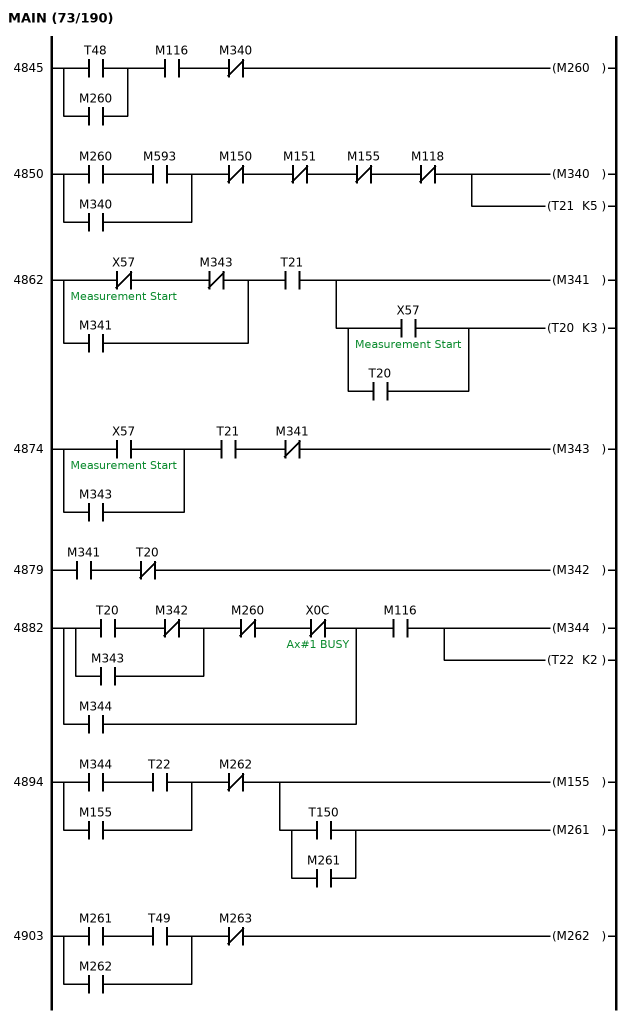
[picture p72: ladder of MAIN, rungs at steps 4845 to 4903]
4845  LD      T48
      OR      M260
      AND     M116
      ANI     M340
      OUT     M260
4850  LD      M260
      AND     M593
      OR      M340
      ANI     M150
      ANI     M151
      ANI     M155
      ANI     M118
      OUT     M340
      OUT     T21 K5
4862  LDI     X57  ; Measurement Start
      ANI     M343
      OR      M341
      AND     T21
      OUT     M341
      LD      X57  ; Measurement Start
      OR      T20
      ANB
      OUT     T20 K3
4874  LD      X57  ; Measurement Start
      OR      M343
      AND     T21
      ANI     M341
      OUT     M343
4879  LD      M341
      ANI     T20
      OUT     M342
4882  LD      T20
      ANI     M342
      OR      M343
      ANI     M260
      ANI     X0C  ; Ax#1 BUSY
      OR      M344
      AND     M116
      OUT     M344
      OUT     T22 K2
4894  LD      M344
      AND     T22
      OR      M155
      ANI     M262
      OUT     M155
      LD      T150
      OR      M261
      ANB
      OUT     M261
4903  LD      M261
      AND     T49
      OR      M262
      ANI     M263
      OUT     M262
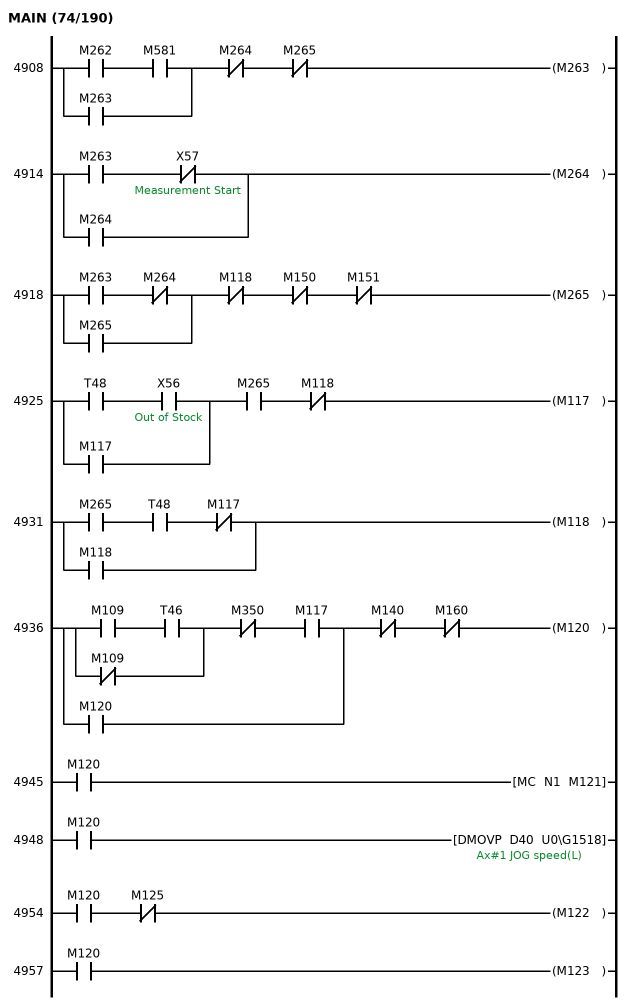
4908  LD      M262
      AND     M581
      OR      M263
      ANI     M264
      ANI     M265
      OUT     M263
4914  LD      M263
      ANI     X57  ; Measurement Start
      OR      M264
      OUT     M264
4918  LD      M263
      ANI     M264
      OR      M265
      ANI     M118
      ANI     M150
      ANI     M151
      OUT     M265
4925  LD      T48
      AND     X56  ; Out of Stock
      OR      M117
      AND     M265
      ANI     M118
      OUT     M117
4931  LD      M265
      AND     T48
      ANI     M117
      OR      M118
      OUT     M118
4936  LD      M109
      AND     T46
      ORI     M109
      ANI     M350
      AND     M117
      OR      M120
      ANI     M140
      ANI     M160
      OUT     M120
4945  LD      M120
      MC      N1 M121
4948  LD      M120
      DMOVP   D40 U0\G1518
4954  LD      M120
      ANI     M125
      OUT     M122
4957  LD      M120
      OUT     M123
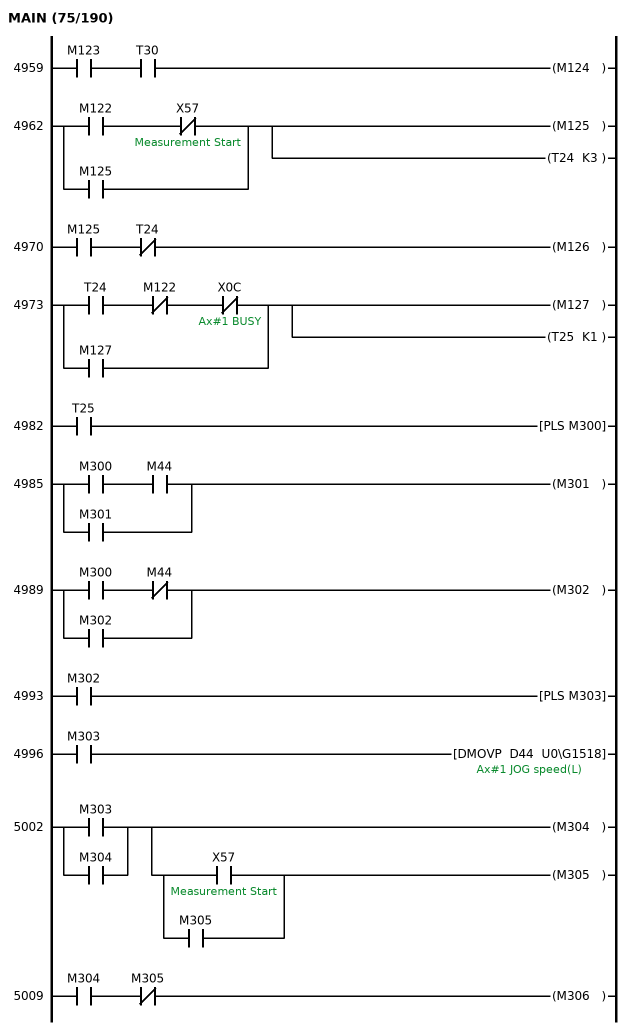
4959  LD      M123
      AND     T30
      OUT     M124
4962  LD      M122
      ANI     X57  ; Measurement Start
      OR      M125
      OUT     M125
      OUT     T24 K3
4970  LD      M125
      ANI     T24
      OUT     M126
4973  LD      T24
      ANI     M122
      ANI     X0C  ; Ax#1 BUSY
      OR      M127
      OUT     M127
      OUT     T25 K1
4982  LD      T25
      PLS     M300
4985  LD      M300
      AND     M44
      OR      M301
      OUT     M301
4989  LD      M300
      ANI     M44
      OR      M302
      OUT     M302
4993  LD      M302
      PLS     M303
4996  LD      M303
      DMOVP   D44 U0\G1518
5002  LD      M303
      OR      M304
      OUT     M304
      LD      X57  ; Measurement Start
      OR      M305
      ANB
      OUT     M305
5009  LD      M304
      ANI     M305
      OUT     M306
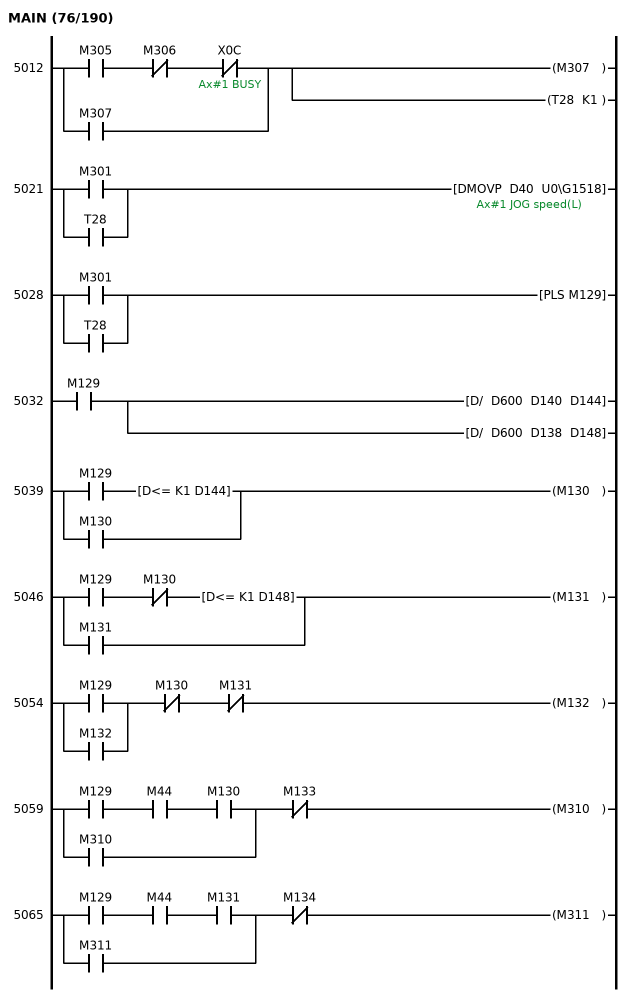
5012  LD      M305
      ANI     M306
      ANI     X0C  ; Ax#1 BUSY
      OR      M307
      OUT     M307
      OUT     T28 K1
5021  LD      M301
      OR      T28
      DMOVP   D40 U0\G1518
5028  LD      M301
      OR      T28
      PLS     M129
5032  LD      M129
      D/      D600 D140 D144
      D/      D600 D138 D148
5039  LD      M129
      ANDD<=  K1 D144
      OR      M130
      OUT     M130
5046  LD      M129
      ANI     M130
      ANDD<=  K1 D148
      OR      M131
      OUT     M131
5054  LD      M129
      OR      M132
      ANI     M130
      ANI     M131
      OUT     M132
5059  LD      M129
      AND     M44
      AND     M130
      OR      M310
      ANI     M133
      OUT     M310
5065  LD      M129
      AND     M44
      AND     M131
      OR      M311
      ANI     M134
      OUT     M311
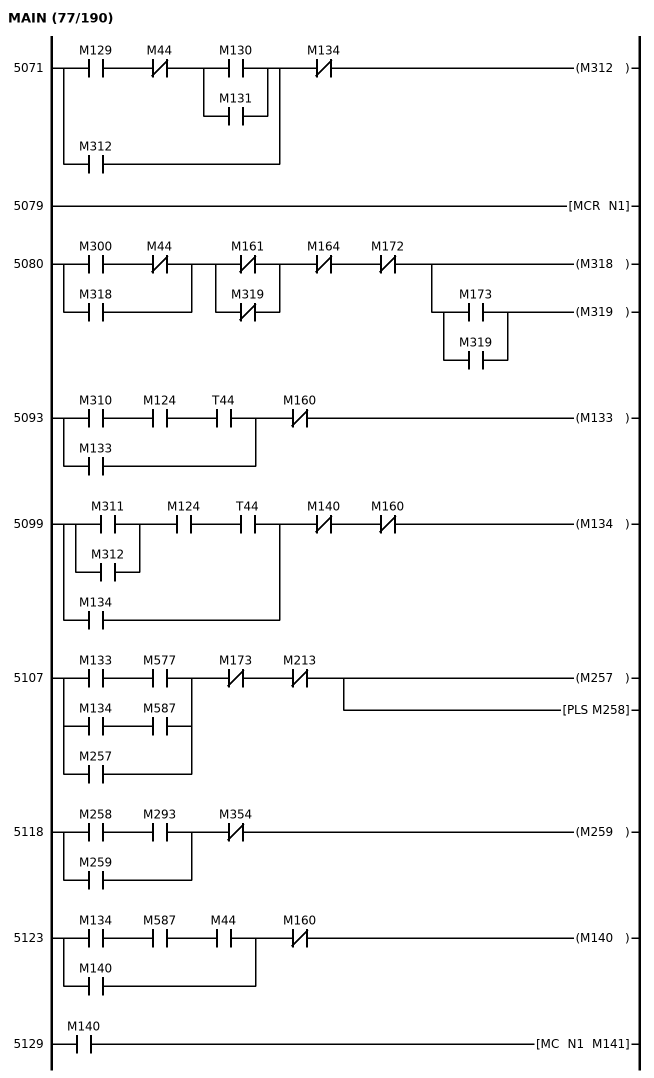
5071  LD      M129
      ANI     M44
      LD      M130
      OR      M131
      ANB
      OR      M312
      ANI     M134
      OUT     M312
5079  MCR     N1
5080  LD      M300
      ANI     M44
      OR      M318
      LDI     M161
      ORI     M319
      ANB
      ANI     M164
      ANI     M172
      OUT     M318
      LD      M173
      OR      M319
      ANB
      OUT     M319
5093  LD      M310
      AND     M124
      AND     T44
      OR      M133
      ANI     M160
      OUT     M133
5099  LD      M311
      OR      M312
      AND     M124
      AND     T44
      OR      M134
      ANI     M140
      ANI     M160
      OUT     M134
5107  LD      M133
      AND     M577
      LD      M134
      AND     M587
      ORB
      OR      M257
      ANI     M173
      ANI     M213
      OUT     M257
      PLS     M258
5118  LD      M258
      AND     M293
      OR      M259
      ANI     M354
      OUT     M259
5123  LD      M134
      AND     M587
      AND     M44
      OR      M140
      ANI     M160
      OUT     M140
5129  LD      M140
      MC      N1 M141
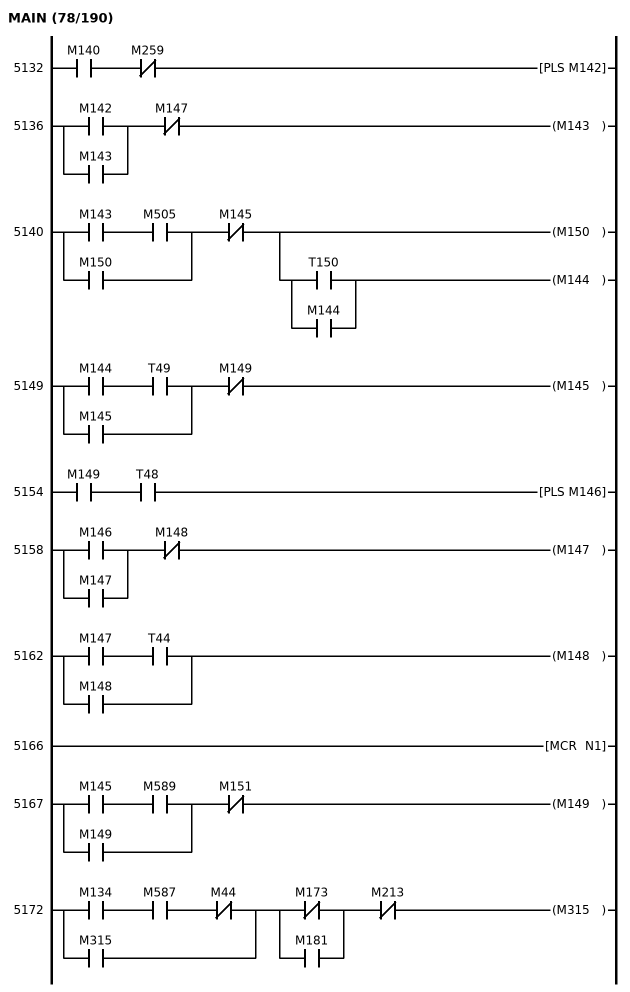
5132  LD      M140
      ANI     M259
      PLS     M142
5136  LD      M142
      OR      M143
      ANI     M147
      OUT     M143
5140  LD      M143
      AND     M505
      OR      M150
      ANI     M145
      OUT     M150
      LD      T150
      OR      M144
      ANB
      OUT     M144
5149  LD      M144
      AND     T49
      OR      M145
      ANI     M149
      OUT     M145
5154  LD      M149
      AND     T48
      PLS     M146
5158  LD      M146
      OR      M147
      ANI     M148
      OUT     M147
5162  LD      M147
      AND     T44
      OR      M148
      OUT     M148
5166  MCR     N1
5167  LD      M145
      AND     M589
      OR      M149
      ANI     M151
      OUT     M149
5172  LD      M134
      AND     M587
      ANI     M44
      OR      M315
      LDI     M173
      OR      M181
      ANB
      ANI     M213
      OUT     M315
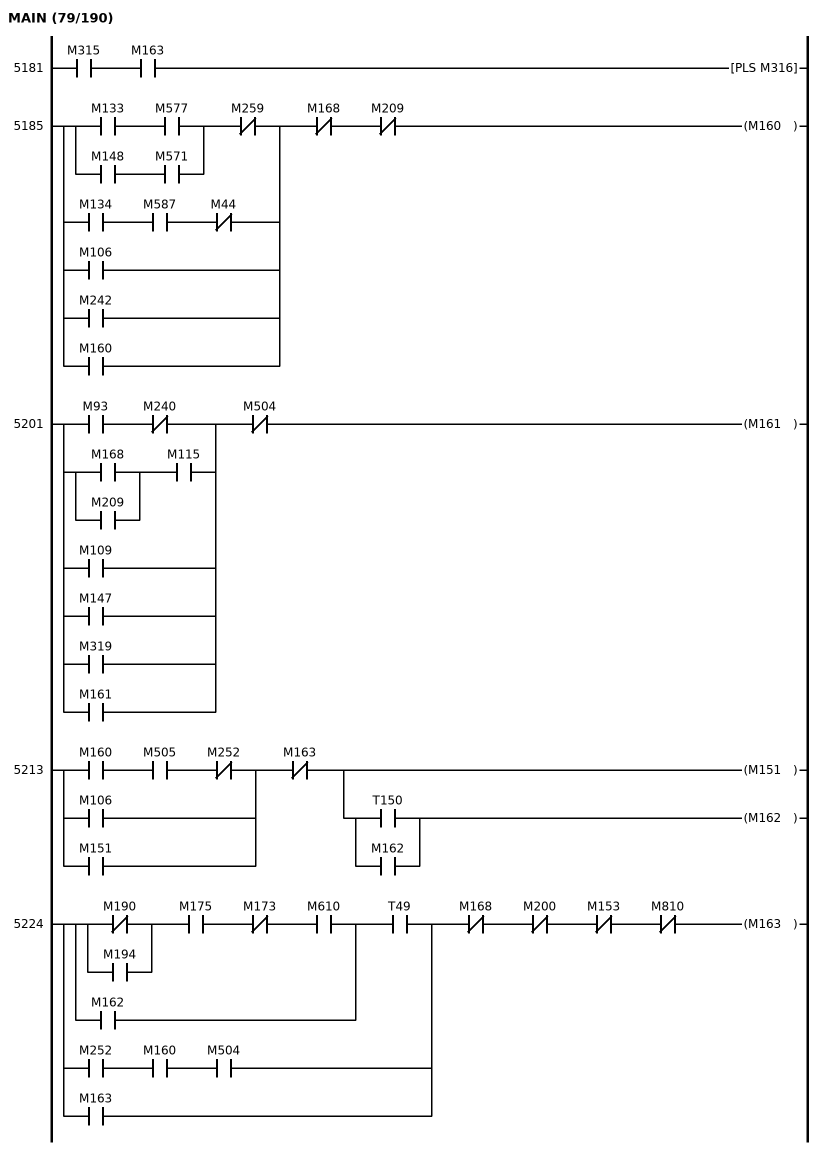
5181  LD      M315
      AND     M163
      PLS     M316
5185  LD      M133
      AND     M577
      LD      M148
      AND     M571
      ORB
      ANI     M259
      LD      M134
      AND     M587
      ANI     M44
      ORB
      OR      M106
      OR      M242
      OR      M160
      ANI     M168
      ANI     M209
      OUT     M160
5201  LD      M93
      ANI     M240
      LD      M168
      OR      M209
      AND     M115
      ORB
      OR      M109
      OR      M147
      OR      M319
      OR      M161
      ANI     M504
      OUT     M161
5213  LD      M160
      AND     M505
      ANI     M252
      OR      M106
      OR      M151
      ANI     M163
      OUT     M151
      LD      T150
      OR      M162
      ANB
      OUT     M162
5224  LDI     M190
      OR      M194
      AND     M175
      ANI     M173
      AND     M610
      OR      M162
      AND     T49
      LD      M252
      AND     M160
      AND     M504
      ORB
      OR      M163
      ANI     M168
      ANI     M200
      ANI     M153
      ANI     M810
      OUT     M163
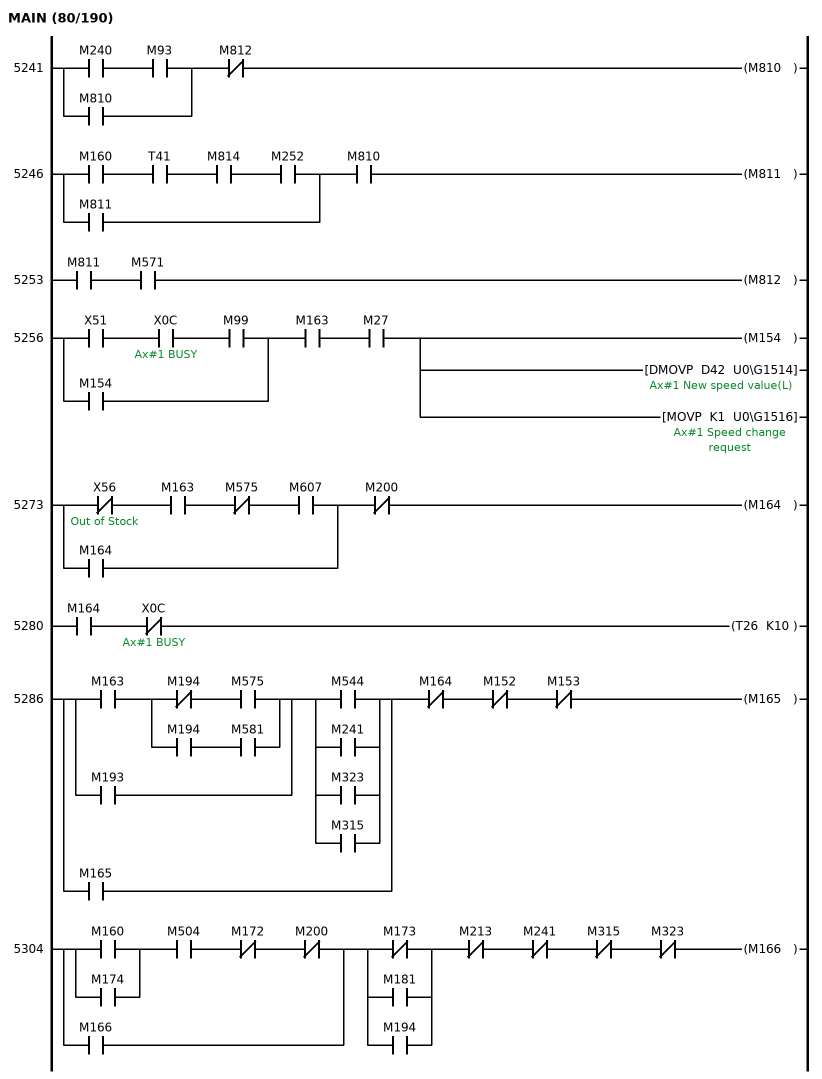
5241  LD      M240
      AND     M93
      OR      M810
      ANI     M812
      OUT     M810
5246  LD      M160
      AND     T41
      AND     M814
      AND     M252
      OR      M811
      AND     M810
      OUT     M811
5253  LD      M811
      AND     M571
      OUT     M812
5256  LD      X51
      AND     X0C  ; Ax#1 BUSY
      AND     M99
      OR      M154
      AND     M163
      AND     M27
      OUT     M154
      DMOVP   D42 U0\G1514  ; Ax#1 New speed value(L)
      MOVP    K1 U0\G1516  ; Ax#1 Speed change request
5273  LDI     X56  ; Out of Stock
      AND     M163
      ANI     M575
      AND     M607
      OR      M164
      ANI     M200
      OUT     M164
5280  LD      M164
      ANI     X0C  ; Ax#1 BUSY
      OUT     T26 K10
5286  LD      M163
      LDI     M194
      AND     M575
      LD      M194
      AND     M581
      ORB
      ANB
      OR      M193
      LD      M544
      OR      M241
      OR      M323
      OR      M315
      ANB
      OR      M165
      ANI     M164
      ANI     M152
      ANI     M153
      OUT     M165
5304  LD      M160
      OR      M174
      AND     M504
      ANI     M172
      ANI     M200
      OR      M166
      LDI     M173
      OR      M181
      OR      M194
      ANB
      ANI     M213
      ANI     M241
      ANI     M315
      ANI     M323
      OUT     M166
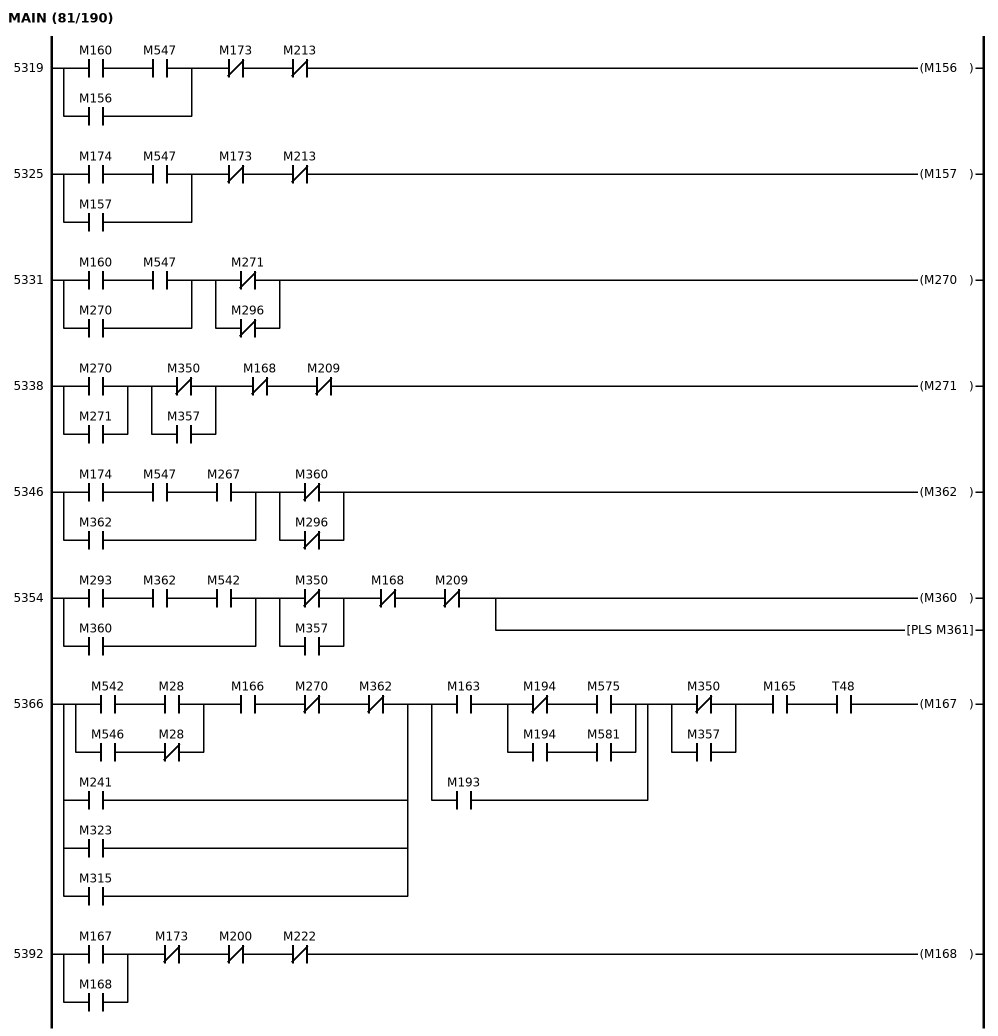
5319  LD      M160
      AND     M547
      OR      M156
      ANI     M173
      ANI     M213
      OUT     M156
5325  LD      M174
      AND     M547
      OR      M157
      ANI     M173
      ANI     M213
      OUT     M157
5331  LD      M160
      AND     M547
      OR      M270
      LDI     M271
      ORI     M296
      ANB
      OUT     M270
5338  LD      M270
      OR      M271
      LDI     M350
      OR      M357
      ANB
      ANI     M168
      ANI     M209
      OUT     M271
5346  LD      M174
      AND     M547
      AND     M267
      OR      M362
      LDI     M360
      ORI     M296
      ANB
      OUT     M362
5354  LD      M293
      AND     M362
      AND     M542
      OR      M360
      LDI     M350
      OR      M357
      ANB
      ANI     M168
      ANI     M209
      OUT     M360
      PLS     M361
5366  LD      M542
      AND     M28
      LD      M546
      ANI     M28
      ORB
      AND     M166
      ANI     M270
      ANI     M362
      OR      M241
      OR      M323
      OR      M315
      LD      M163
      LDI     M194
      AND     M575
      LD      M194
      AND     M581
      ORB
      ANB
      OR      M193
      ANB
      LDI     M350
      OR      M357
      ANB
      AND     M165
      AND     T48
      OUT     M167
5392  LD      M167
      OR      M168
      ANI     M173
      ANI     M200
      ANI     M222
      OUT     M168
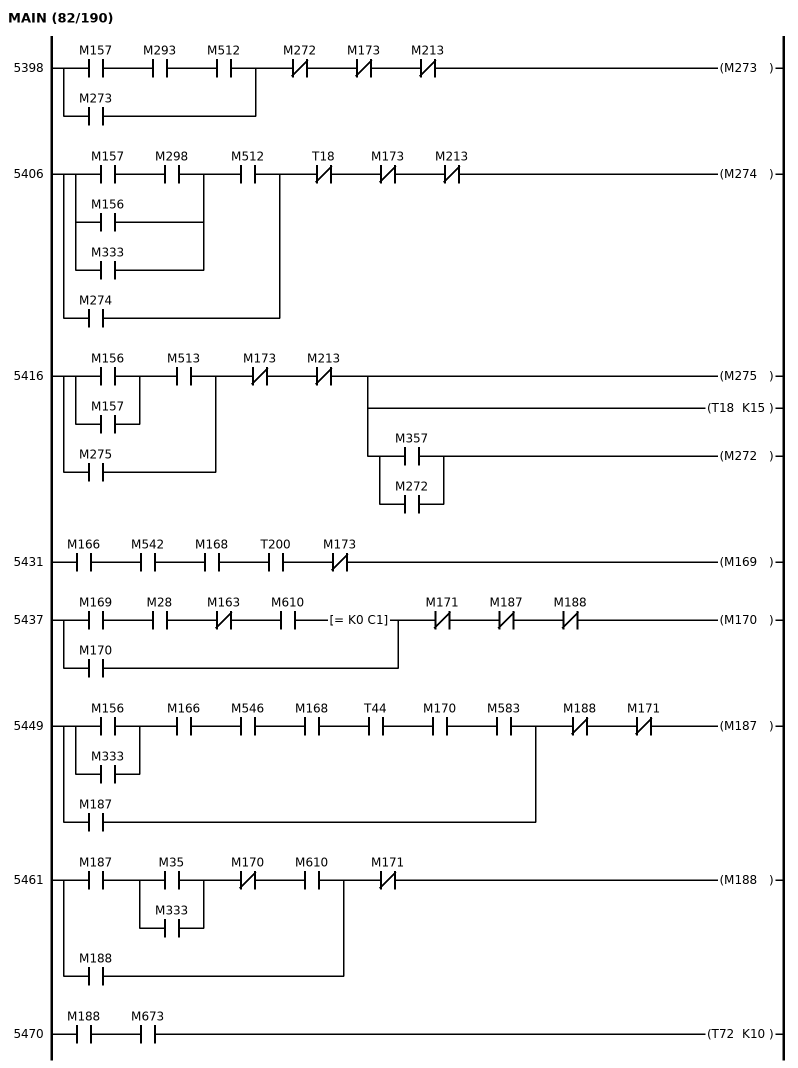
5398  LD      M157
      AND     M293
      AND     M512
      OR      M273
      ANI     M272
      ANI     M173
      ANI     M213
      OUT     M273
5406  LD      M157
      AND     M298
      OR      M156
      OR      M333
      AND     M512
      OR      M274
      ANI     T18
      ANI     M173
      ANI     M213
      OUT     M274
5416  LD      M156
      OR      M157
      AND     M513
      OR      M275
      ANI     M173
      ANI     M213
      OUT     M275
      OUT     T18 K15
      LD      M357
      OR      M272
      ANB
      OUT     M272
5431  LD      M166
      AND     M542
      AND     M168
      AND     T200
      ANI     M173
      OUT     M169
5437  LD      M169
      AND     M28
      ANI     M163
      AND     M610
      AND=    K0 C1
      OR      M170
      ANI     M171
      ANI     M187
      ANI     M188
      OUT     M170
5449  LD      M156
      OR      M333
      AND     M166
      AND     M546
      AND     M168
      AND     T44
      AND     M170
      AND     M583
      OR      M187
      ANI     M188
      ANI     M171
      OUT     M187
5461  LD      M187
      LD      M35
      OR      M333
      ANB
      ANI     M170
      AND     M610
      OR      M188
      ANI     M171
      OUT     M188
5470  LD      M188
      AND     M673
      OUT     T72 K10
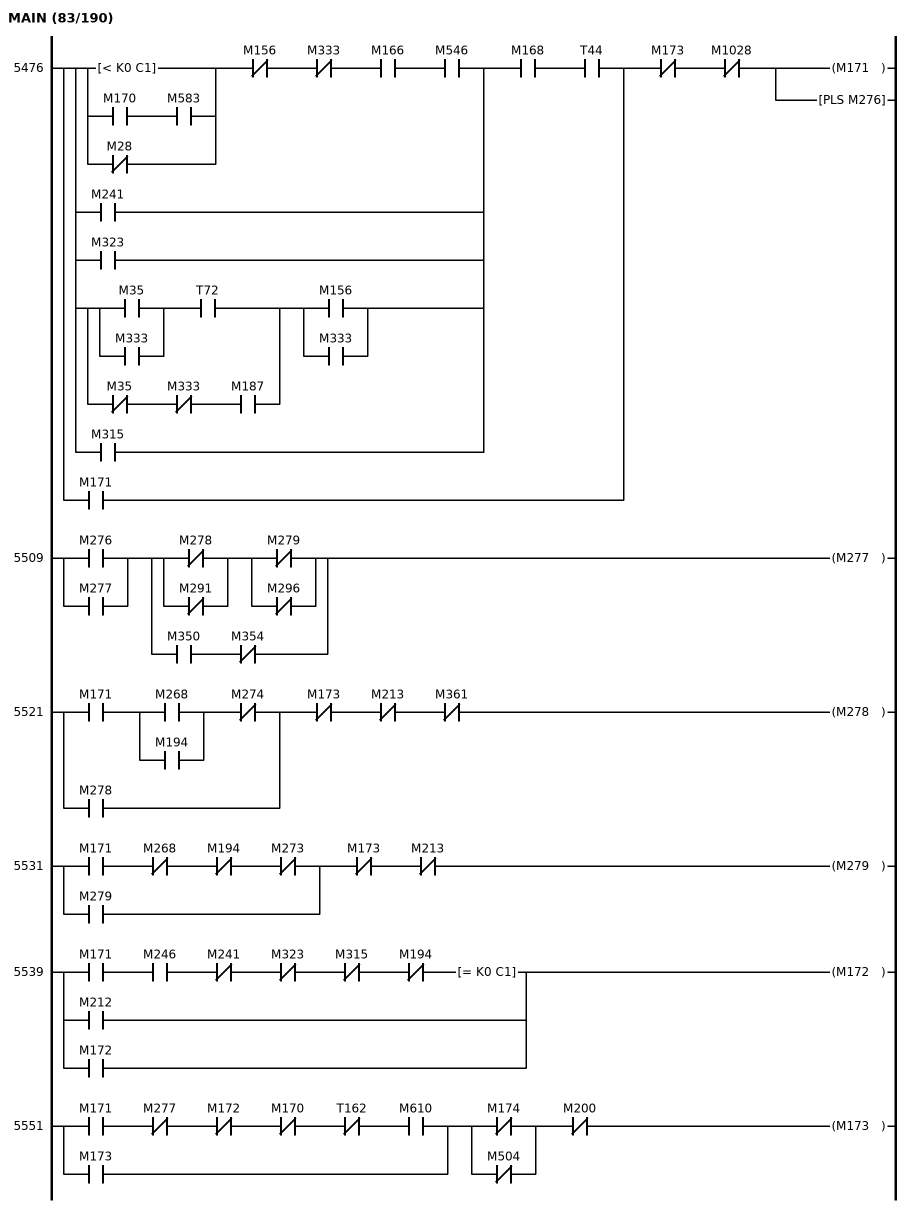
5476  LD<     K0 C1
      LD      M170
      AND     M583
      ORB
      ORI     M28
      ANI     M156
      ANI     M333
      AND     M166
      AND     M546
      OR      M241
      OR      M323
      LD      M35
      OR      M333
      AND     T72
      LDI     M35
      ANI     M333
      AND     M187
      ORB
      LD      M156
      OR      M333
      ANB
      ORB
      OR      M315
      AND     M168
      AND     T44
      OR      M171
      ANI     M173
      ANI     M1028
      OUT     M171
      PLS     M276
5509  LD      M276
      OR      M277
      LDI     M278
      ORI     M291
      LDI     M279
      ORI     M296
      ANB
      LD      M350
      ANI     M354
      ORB
      ANB
      OUT     M277
5521  LD      M171
      LD      M268
      OR      M194
      ANB
      ANI     M274
      OR      M278
      ANI     M173
      ANI     M213
      ANI     M361
      OUT     M278
5531  LD      M171
      ANI     M268
      ANI     M194
      ANI     M273
      OR      M279
      ANI     M173
      ANI     M213
      OUT     M279
5539  LD      M171
      AND     M246
      ANI     M241
      ANI     M323
      ANI     M315
      ANI     M194
      AND=    K0 C1
      OR      M212
      OR      M172
      OUT     M172
5551  LD      M171
      ANI     M277
      ANI     M172
      ANI     M170
      ANI     T162
      AND     M610
      OR      M173
      LDI     M174
      ORI     M504
      ANB
      ANI     M200
      OUT     M173
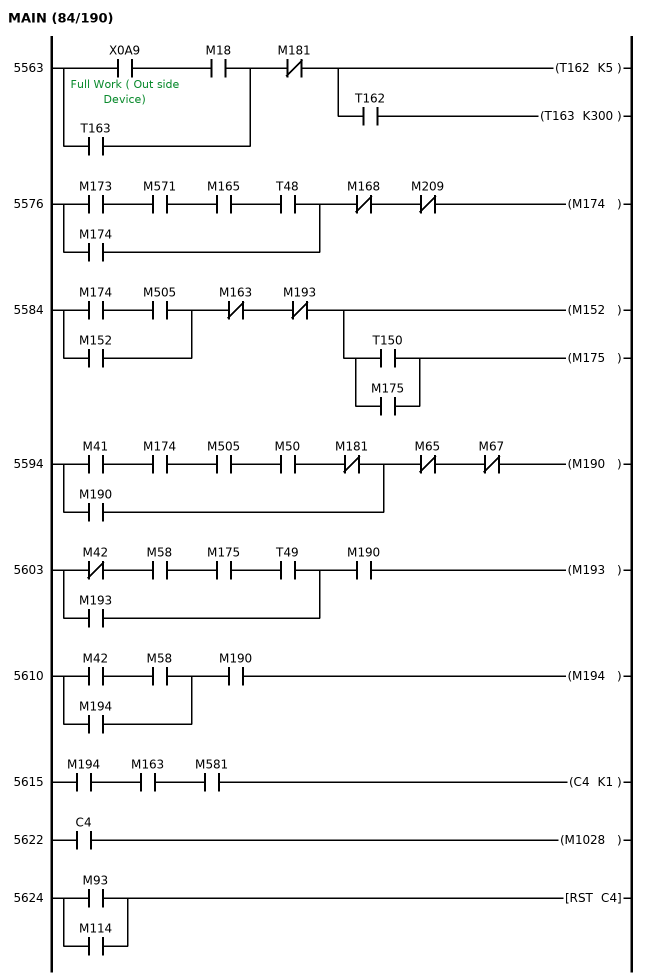
5563  LD      X0A9  ; Full Work ( Out side Device)
      AND     M18
      OR      T163
      ANI     M181
      OUT     T162 K5
      AND     T162
      OUT     T163 K300
5576  LD      M173
      AND     M571
      AND     M165
      AND     T48
      OR      M174
      ANI     M168
      ANI     M209
      OUT     M174
5584  LD      M174
      AND     M505
      OR      M152
      ANI     M163
      ANI     M193
      OUT     M152
      LD      T150
      OR      M175
      ANB
      OUT     M175
5594  LD      M41
      AND     M174
      AND     M505
      AND     M50
      ANI     M181
      OR      M190
      ANI     M65
      ANI     M67
      OUT     M190
5603  LDI     M42
      AND     M58
      AND     M175
      AND     T49
      OR      M193
      AND     M190
      OUT     M193
5610  LD      M42
      AND     M58
      OR      M194
      AND     M190
      OUT     M194
5615  LD      M194
      AND     M163
      AND     M581
      OUT     C4 K1
5622  LD      C4
      OUT     M1028
5624  LD      M93
      OR      M114
      RST     C4
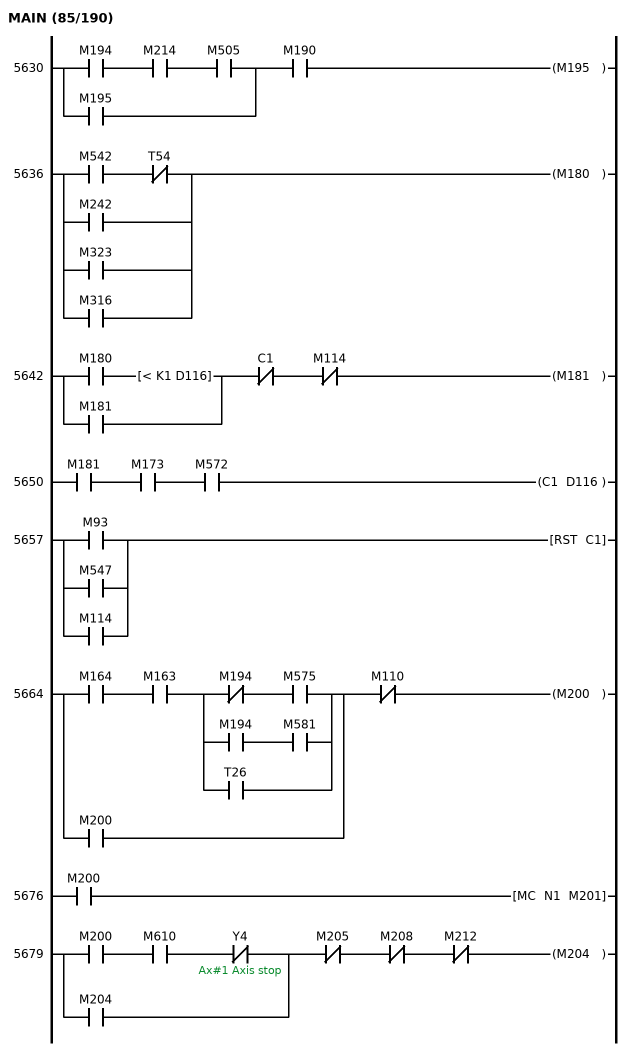
5630  LD      M194
      AND     M214
      AND     M505
      OR      M195
      AND     M190
      OUT     M195
5636  LD      M542
      ANI     T54
      OR      M242
      OR      M323
      OR      M316
      OUT     M180
5642  LD      M180
      AND<    K1 D116
      OR      M181
      ANI     C1
      ANI     M114
      OUT     M181
5650  LD      M181
      AND     M173
      AND     M572
      OUT     C1 D116
5657  LD      M93
      OR      M547
      OR      M114
      RST     C1
5664  LD      M164
      AND     M163
      LDI     M194
      AND     M575
      LD      M194
      AND     M581
      ORB
      OR      T26
      ANB
      OR      M200
      ANI     M110
      OUT     M200
5676  LD      M200
      MC      N1 M201
5679  LD      M200
      AND     M610
      ANI     Y4  ; Ax#1 Axis stop
      OR      M204
      ANI     M205
      ANI     M208
      ANI     M212
      OUT     M204
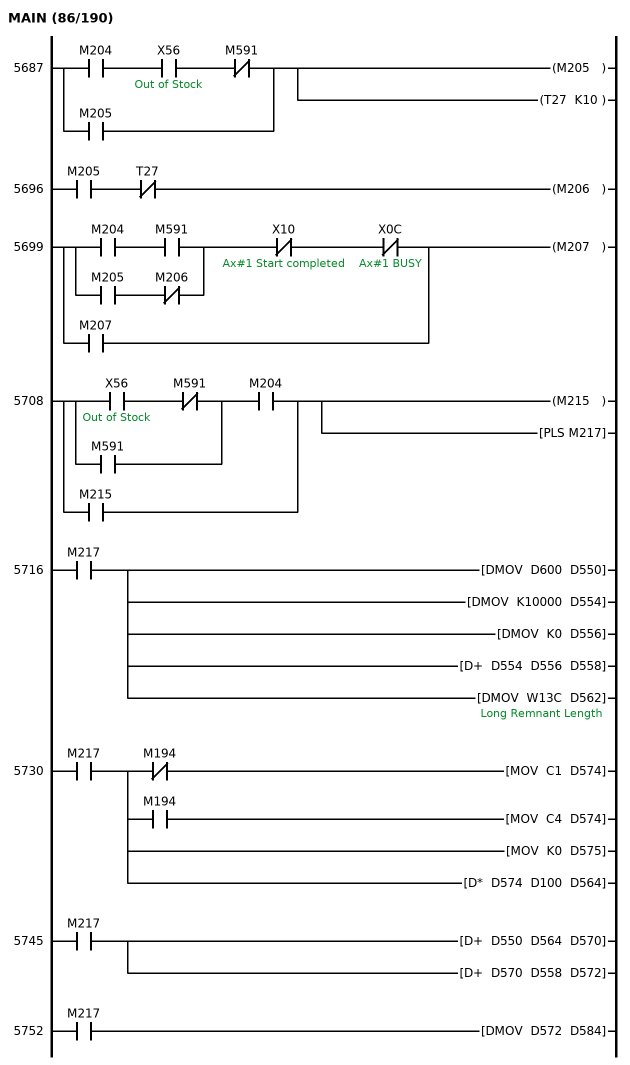
5687  LD      M204
      AND     X56  ; Out of Stock
      ANI     M591
      OR      M205
      OUT     M205
      OUT     T27 K10
5696  LD      M205
      ANI     T27
      OUT     M206
5699  LD      M204
      AND     M591
      LD      M205
      ANI     M206
      ORB
      ANI     X10  ; Ax#1 Start completed
      ANI     X0C  ; Ax#1 BUSY
      OR      M207
      OUT     M207
5708  LD      X56  ; Out of Stock
      ANI     M591
      OR      M591
      AND     M204
      OR      M215
      OUT     M215
      PLS     M217
5716  LD      M217
      DMOV    D600 D550
      DMOV    K10000 D554
      DMOV    K0 D556
      D+      D554 D556 D558
      DMOV    W13C D562  ; Long Remnant Length
5730  LD      M217
      MPS
      ANI     M194
      MOV     C1 D574
      MRD
      AND     M194
      MOV     C4 D574
      MPP
      MOV     K0 D575
      D*      D574 D100 D564
5745  LD      M217
      D+      D550 D564 D570
      D+      D570 D558 D572
5752  LD      M217
      DMOV    D572 D584
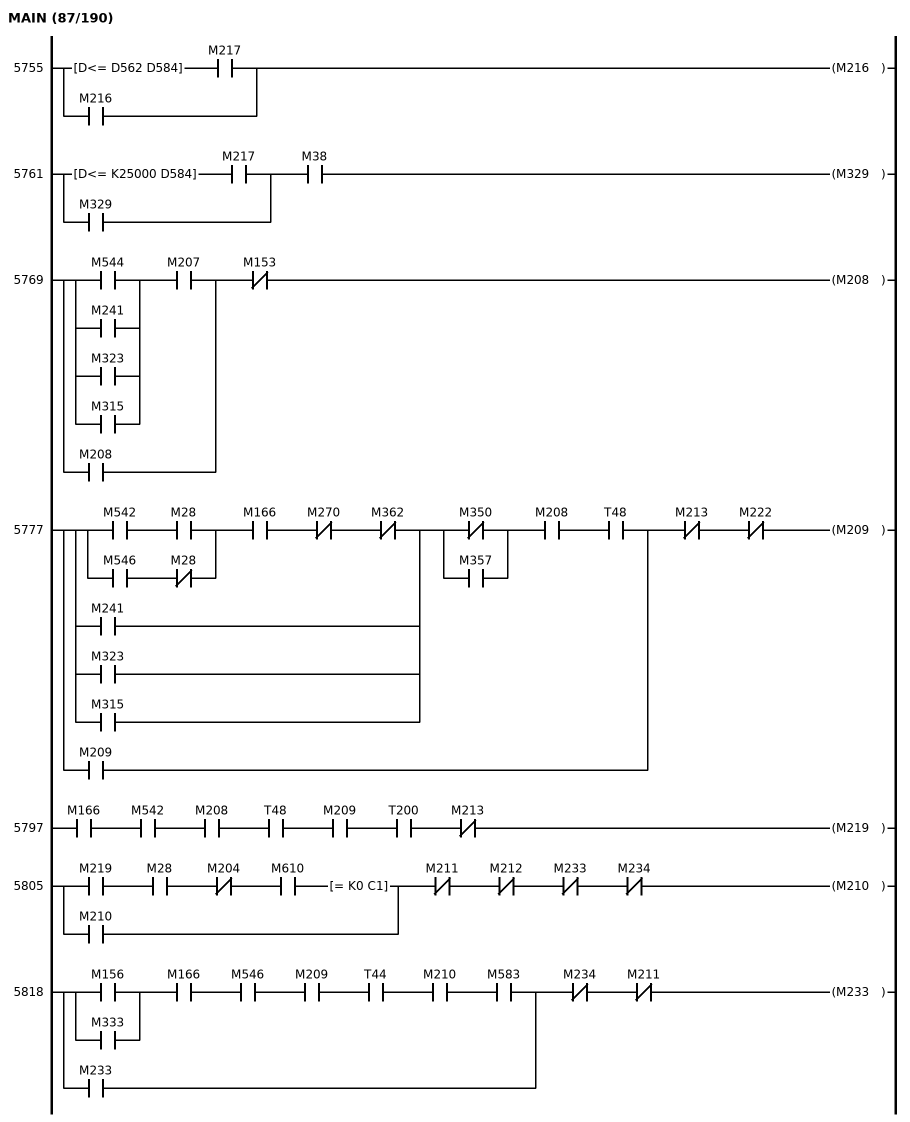
5755  LDD<=   D562 D584
      AND     M217
      OR      M216
      OUT     M216
5761  LDD<=   K25000 D584
      AND     M217
      OR      M329
      AND     M38
      OUT     M329
5769  LD      M544
      OR      M241
      OR      M323
      OR      M315
      AND     M207
      OR      M208
      ANI     M153
      OUT     M208
5777  LD      M542
      AND     M28
      LD      M546
      ANI     M28
      ORB
      AND     M166
      ANI     M270
      ANI     M362
      OR      M241
      OR      M323
      OR      M315
      LDI     M350
      OR      M357
      ANB
      AND     M208
      AND     T48
      OR      M209
      ANI     M213
      ANI     M222
      OUT     M209
5797  LD      M166
      AND     M542
      AND     M208
      AND     T48
      AND     M209
      AND     T200
      ANI     M213
      OUT     M219
5805  LD      M219
      AND     M28
      ANI     M204
      AND     M610
      AND=    K0 C1
      OR      M210
      ANI     M211
      ANI     M212
      ANI     M233
      ANI     M234
      OUT     M210
5818  LD      M156
      OR      M333
      AND     M166
      AND     M546
      AND     M209
      AND     T44
      AND     M210
      AND     M583
      OR      M233
      ANI     M234
      ANI     M211
      OUT     M233
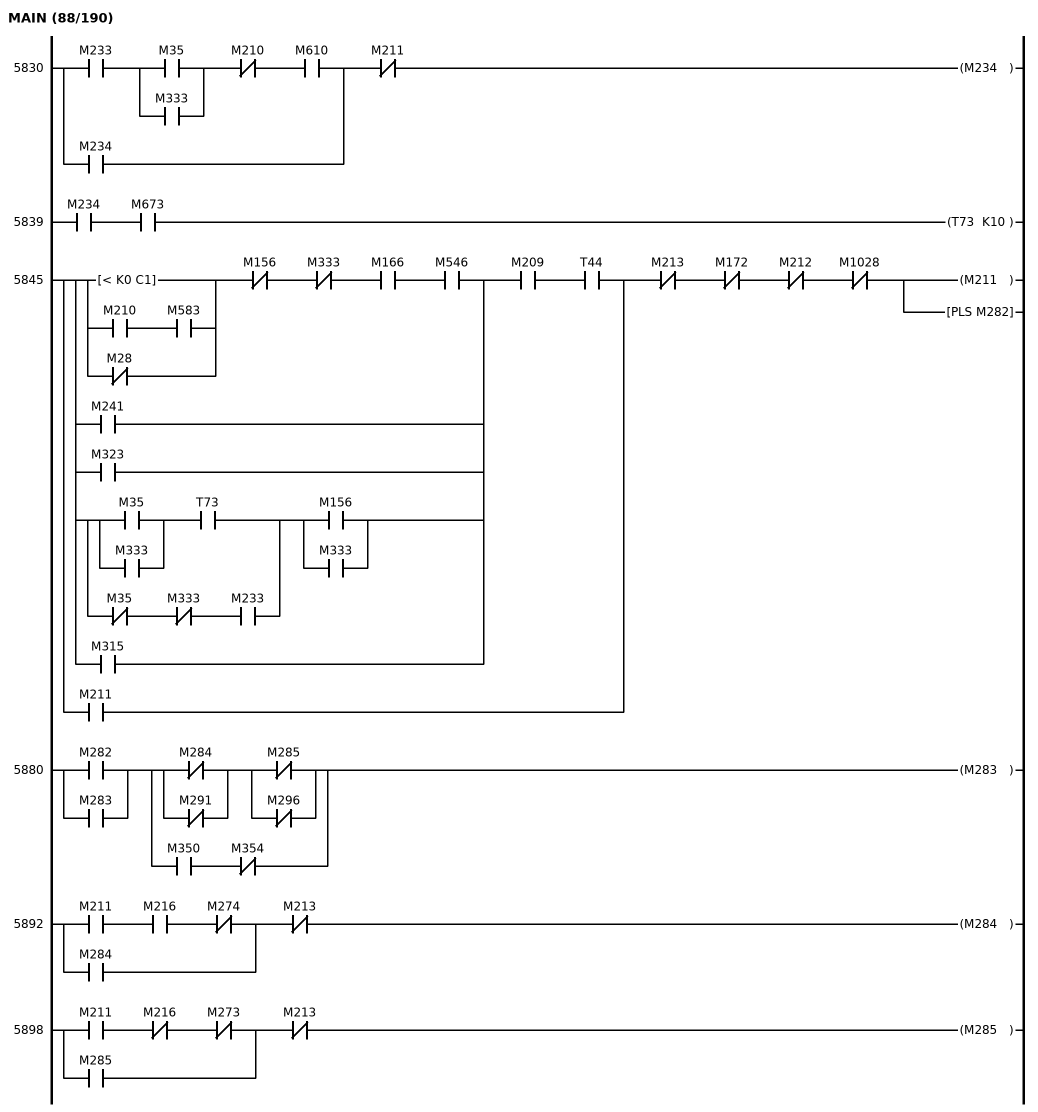
5830  LD      M233
      LD      M35
      OR      M333
      ANB
      ANI     M210
      AND     M610
      OR      M234
      ANI     M211
      OUT     M234
5839  LD      M234
      AND     M673
      OUT     T73 K10
5845  LD<     K0 C1
      LD      M210
      AND     M583
      ORB
      ORI     M28
      ANI     M156
      ANI     M333
      AND     M166
      AND     M546
      OR      M241
      OR      M323
      LD      M35
      OR      M333
      AND     T73
      LDI     M35
      ANI     M333
      AND     M233
      ORB
      LD      M156
      OR      M333
      ANB
      ORB
      OR      M315
      AND     M209
      AND     T44
      OR      M211
      ANI     M213
      ANI     M172
      ANI     M212
      ANI     M1028
      OUT     M211
      PLS     M282
5880  LD      M282
      OR      M283
      LDI     M284
      ORI     M291
      LDI     M285
      ORI     M296
      ANB
      LD      M350
      ANI     M354
      ORB
      ANB
      OUT     M283
5892  LD      M211
      AND     M216
      ANI     M274
      OR      M284
      ANI     M213
      OUT     M284
5898  LD      M211
      ANI     M216
      ANI     M273
      OR      M285
      ANI     M213
      OUT     M285
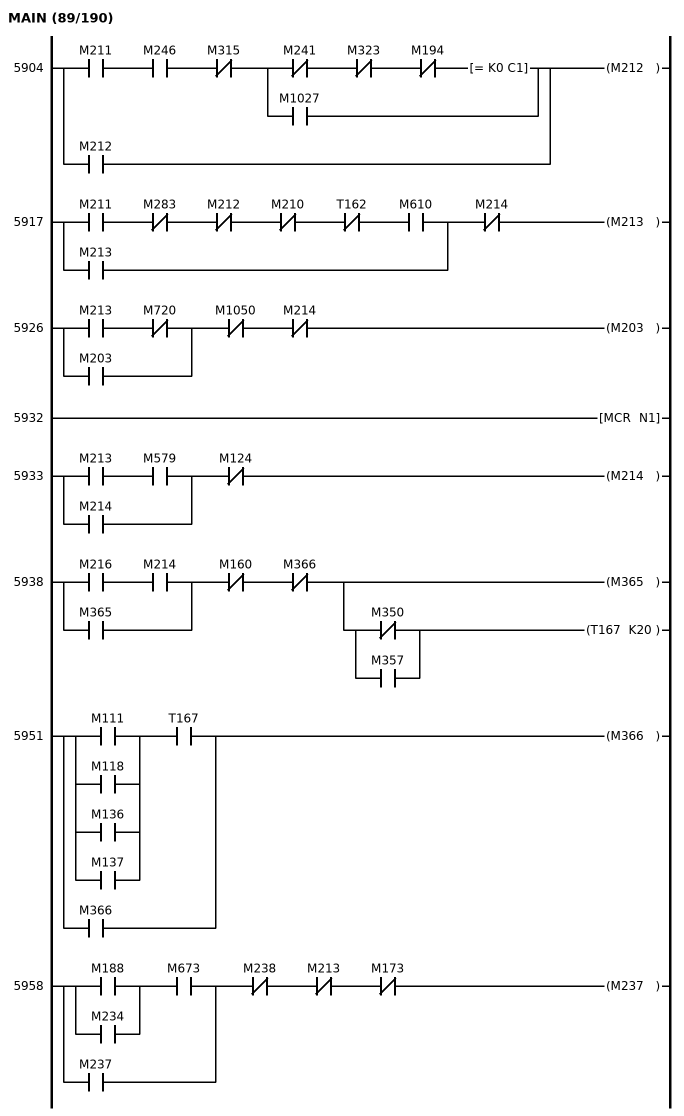
5904  LD      M211
      AND     M246
      ANI     M315
      LDI     M241
      ANI     M323
      ANI     M194
      AND=    K0 C1
      OR      M1027
      ANB
      OR      M212
      OUT     M212
5917  LD      M211
      ANI     M283
      ANI     M212
      ANI     M210
      ANI     T162
      AND     M610
      OR      M213
      ANI     M214
      OUT     M213
5926  LD      M213
      ANI     M720
      OR      M203
      ANI     M1050
      ANI     M214
      OUT     M203
5932  MCR     N1
5933  LD      M213
      AND     M579
      OR      M214
      ANI     M124
      OUT     M214
5938  LD      M216
      AND     M214
      OR      M365
      ANI     M160
      ANI     M366
      OUT     M365
      LDI     M350
      OR      M357
      ANB
      OUT     T167 K20
5951  LD      M111
      OR      M118
      OR      M136
      OR      M137
      AND     T167
      OR      M366
      OUT     M366
5958  LD      M188
      OR      M234
      AND     M673
      OR      M237
      ANI     M238
      ANI     M213
      ANI     M173
      OUT     M237
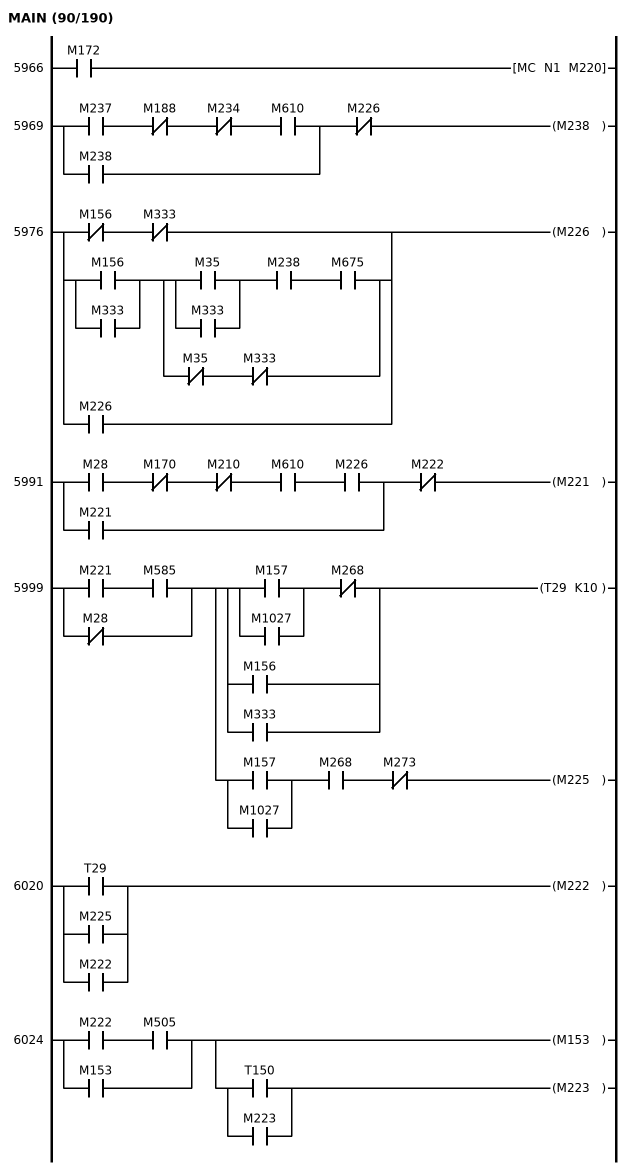
5966  LD      M172
      MC      N1 M220
5969  LD      M237
      ANI     M188
      ANI     M234
      AND     M610
      OR      M238
      ANI     M226
      OUT     M238
5976  LDI     M156
      ANI     M333
      LD      M156
      OR      M333
      LD      M35
      OR      M333
      AND     M238
      AND     M675
      LDI     M35
      ANI     M333
      ORB
      ANB
      ORB
      OR      M226
      OUT     M226
5991  LD      M28
      ANI     M170
      ANI     M210
      AND     M610
      AND     M226
      OR      M221
      ANI     M222
      OUT     M221
5999  LD      M221
      AND     M585
      ORI     M28
      MPS
      LD      M157
      OR      M1027
      ANI     M268
      OR      M156
      OR      M333
      ANB
      OUT     T29 K10
      MPP
      LD      M157
      OR      M1027
      ANB
      AND     M268
      ANI     M273
      OUT     M225
6020  LD      T29
      OR      M225
      OR      M222
      OUT     M222
6024  LD      M222
      AND     M505
      OR      M153
      OUT     M153
      LD      T150
      OR      M223
      ANB
      OUT     M223
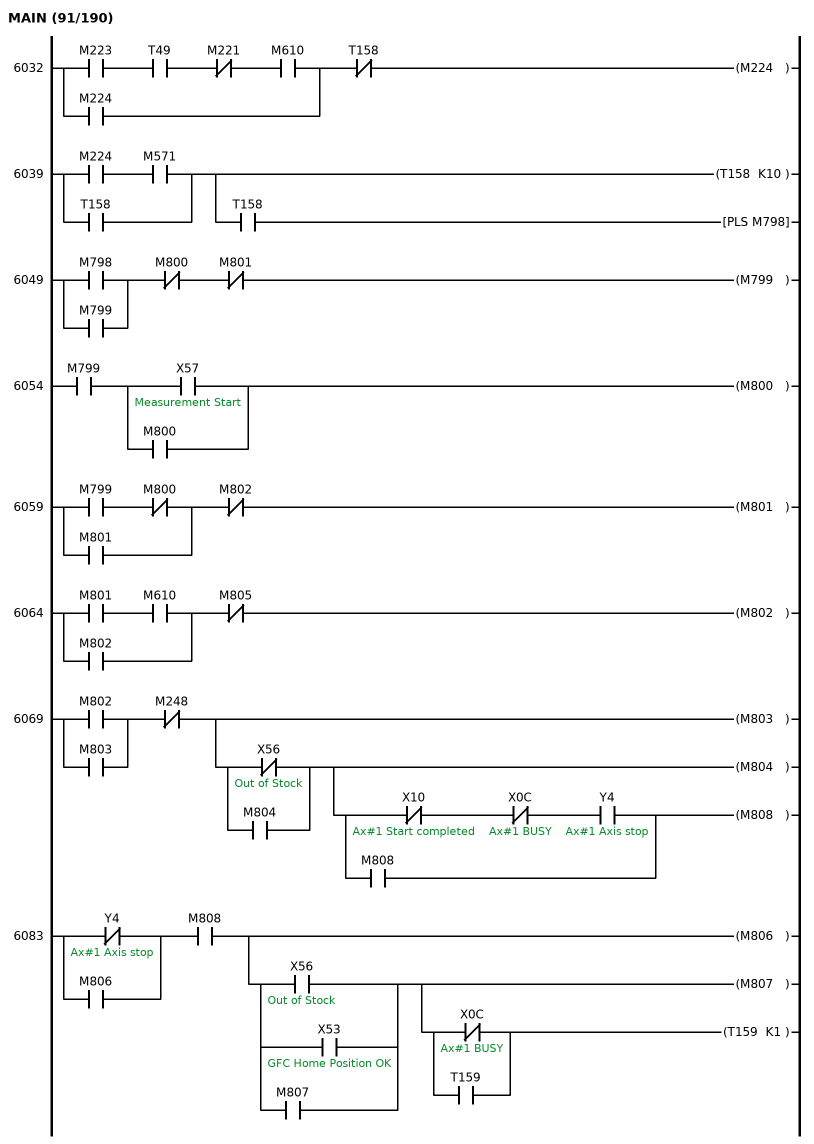
6032  LD      M223
      AND     T49
      ANI     M221
      AND     M610
      OR      M224
      ANI     T158
      OUT     M224
6039  LD      M224
      AND     M571
      OR      T158
      OUT     T158 K10
      AND     T158
      PLS     M798
6049  LD      M798
      OR      M799
      ANI     M800
      ANI     M801
      OUT     M799
6054  LD      M799
      LD      X57  ; Measurement Start
      OR      M800
      ANB
      OUT     M800
6059  LD      M799
      ANI     M800
      OR      M801
      ANI     M802
      OUT     M801
6064  LD      M801
      AND     M610
      OR      M802
      ANI     M805
      OUT     M802
6069  LD      M802
      OR      M803
      ANI     M248
      OUT     M803
      LDI     X56  ; Out of Stock
      OR      M804
      ANB
      OUT     M804
      LDI     X10  ; Ax#1 Start completed
      ANI     X0C  ; Ax#1 BUSY
      AND     Y4  ; Ax#1 Axis stop
      OR      M808
      ANB
      OUT     M808
6083  LDI     Y4  ; Ax#1 Axis stop
      OR      M806
      AND     M808
      OUT     M806
      LD      X56  ; Out of Stock
      OR      X53  ; GFC Home Position OK
      OR      M807
      ANB
      OUT     M807
      LDI     X0C  ; Ax#1 BUSY
      OR      T159
      ANB
      OUT     T159 K1
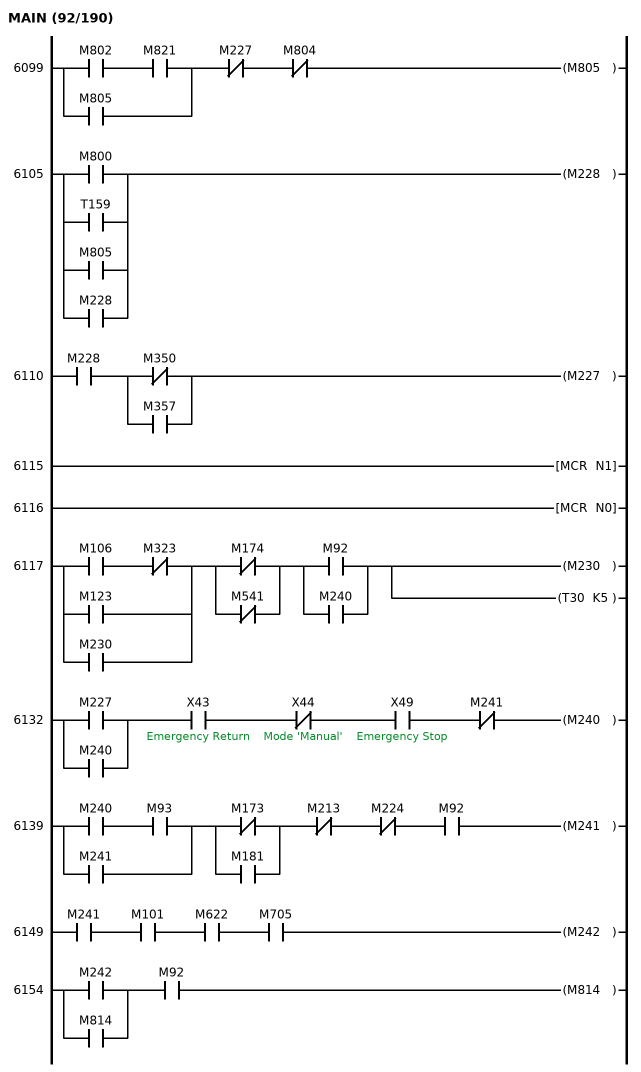
6099  LD      M802
      AND     M821
      OR      M805
      ANI     M227
      ANI     M804
      OUT     M805
6105  LD      M800
      OR      T159
      OR      M805
      OR      M228
      OUT     M228
6110  LD      M228
      LDI     M350
      OR      M357
      ANB
      OUT     M227
6115  MCR     N1
6116  MCR     N0
6117  LD      M106
      ANI     M323
      OR      M123
      OR      M230
      LDI     M174
      ORI     M541
      ANB
      LD      M92
      OR      M240
      ANB
      OUT     M230
      OUT     T30 K5
6132  LD      M227
      OR      M240
      AND     X43  ; Emergency Return
      ANI     X44  ; Mode 'Manual'
      AND     X49  ; Emergency Stop
      ANI     M241
      OUT     M240
6139  LD      M240
      AND     M93
      OR      M241
      LDI     M173
      OR      M181
      ANB
      ANI     M213
      ANI     M224
      AND     M92
      OUT     M241
6149  LD      M241
      AND     M101
      AND     M622
      AND     M705
      OUT     M242
6154  LD      M242
      OR      M814
      AND     M92
      OUT     M814
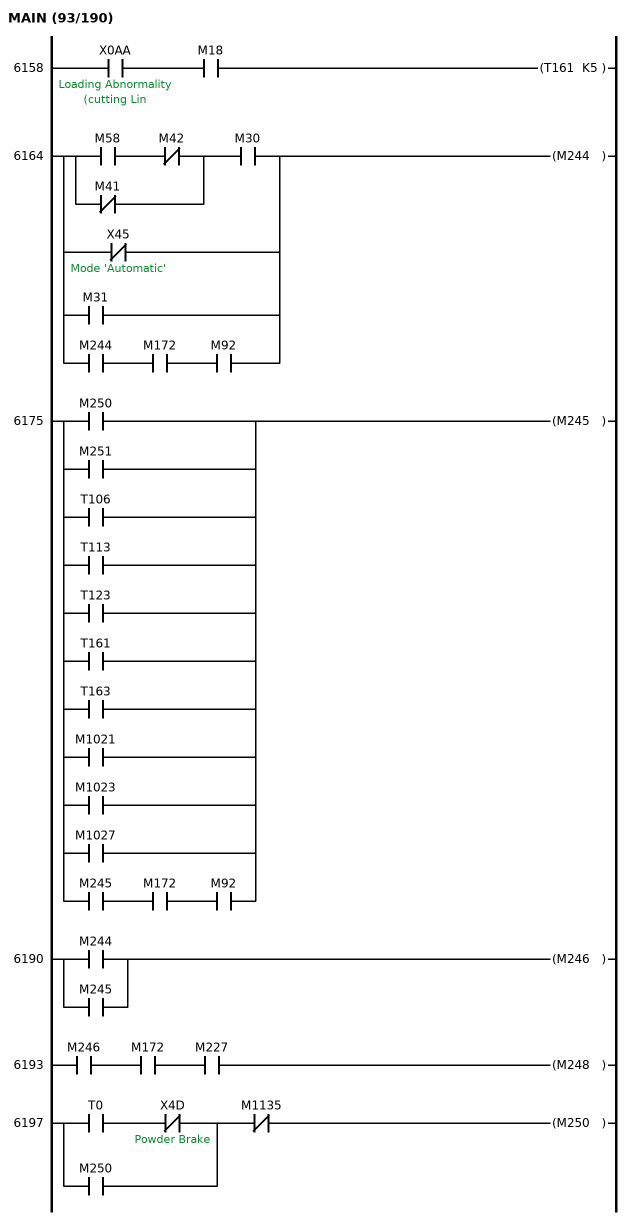
6158  LD      X0AA  ; Loading Abnormality (cutting Lin
      AND     M18
      OUT     T161 K5
6164  LD      M58
      ANI     M42
      ORI     M41
      AND     M30
      ORI     X45  ; Mode 'Automatic'
      OR      M31
      LD      M244
      AND     M172
      AND     M92
      ORB
      OUT     M244
6175  LD      M250
      OR      M251
      OR      T106
      OR      T113
      OR      T123
      OR      T161
      OR      T163
      OR      M1021
      OR      M1023
      OR      M1027
      LD      M245
      AND     M172
      AND     M92
      ORB
      OUT     M245
6190  LD      M244
      OR      M245
      OUT     M246
6193  LD      M246
      AND     M172
      AND     M227
      OUT     M248
6197  LD      T0
      ANI     X4D  ; Powder Brake
      OR      M250
      ANI     M1135
      OUT     M250
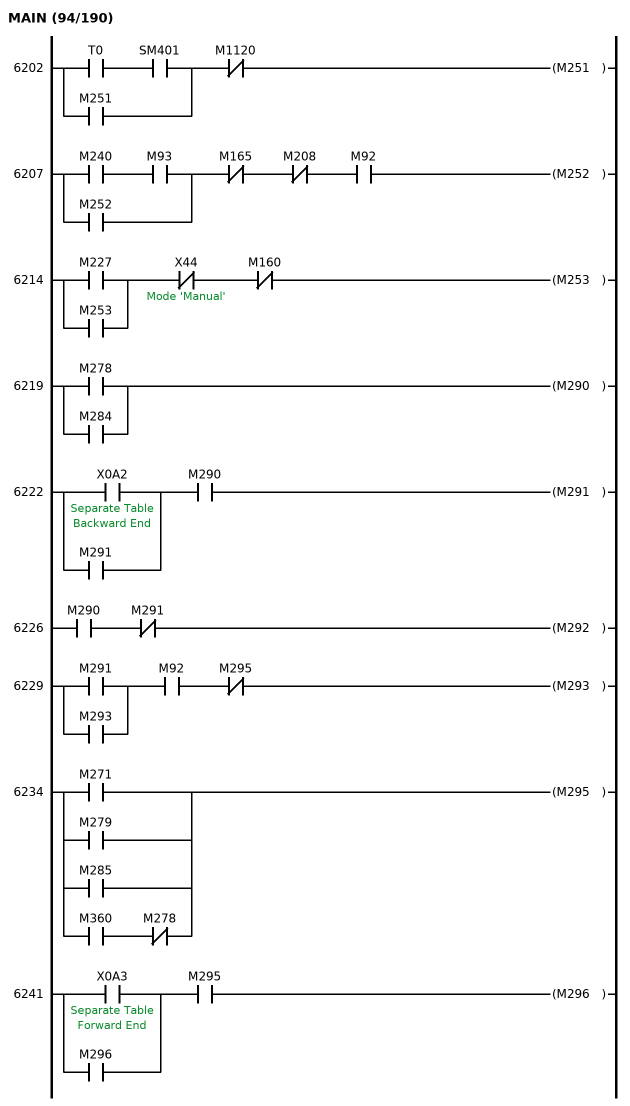
6202  LD      T0
      AND     SM401
      OR      M251
      ANI     M1120
      OUT     M251
6207  LD      M240
      AND     M93
      OR      M252
      ANI     M165
      ANI     M208
      AND     M92
      OUT     M252
6214  LD      M227
      OR      M253
      ANI     X44  ; Mode 'Manual'
      ANI     M160
      OUT     M253
6219  LD      M278
      OR      M284
      OUT     M290
6222  LD      X0A2  ; Separate Table Backward End
      OR      M291
      AND     M290
      OUT     M291
6226  LD      M290
      ANI     M291
      OUT     M292
6229  LD      M291
      OR      M293
      AND     M92
      ANI     M295
      OUT     M293
6234  LD      M271
      OR      M279
      OR      M285
      LD      M360
      ANI     M278
      ORB
      OUT     M295
6241  LD      X0A3  ; Separate Table Forward End
      OR      M296
      AND     M295
      OUT     M296
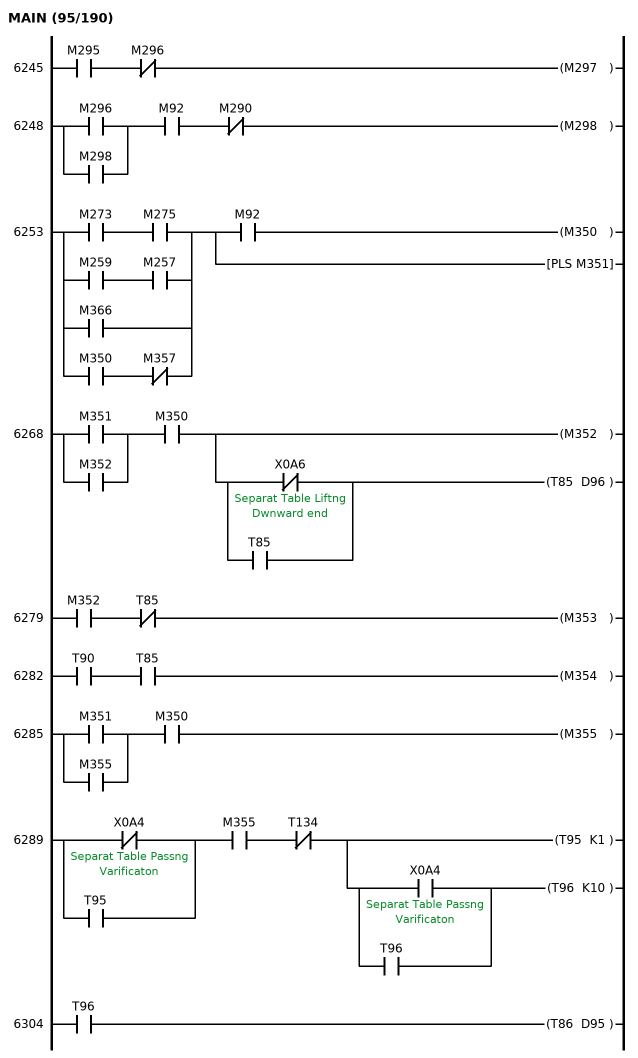
6245  LD      M295
      ANI     M296
      OUT     M297
6248  LD      M296
      OR      M298
      AND     M92
      ANI     M290
      OUT     M298
6253  LD      M273
      AND     M275
      LD      M259
      AND     M257
      ORB
      OR      M366
      LD      M350
      ANI     M357
      ORB
      MPS
      AND     M92
      OUT     M350
      MPP
      PLS     M351
6268  LD      M351
      OR      M352
      AND     M350
      OUT     M352
      LDI     X0A6  ; Separat Table Liftng Dwnward end
      OR      T85
      ANB
      OUT     T85 D96
6279  LD      M352
      ANI     T85
      OUT     M353
6282  LD      T90
      AND     T85
      OUT     M354
6285  LD      M351
      OR      M355
      AND     M350
      OUT     M355
6289  LDI     X0A4  ; Separat Table Passng Varificaton
      OR      T95
      AND     M355
      ANI     T134
      OUT     T95 K1
      LD      X0A4  ; Separat Table Passng Varificaton
      OR      T96
      ANB
      OUT     T96 K10
6304  LD      T96
      OUT     T86 D95
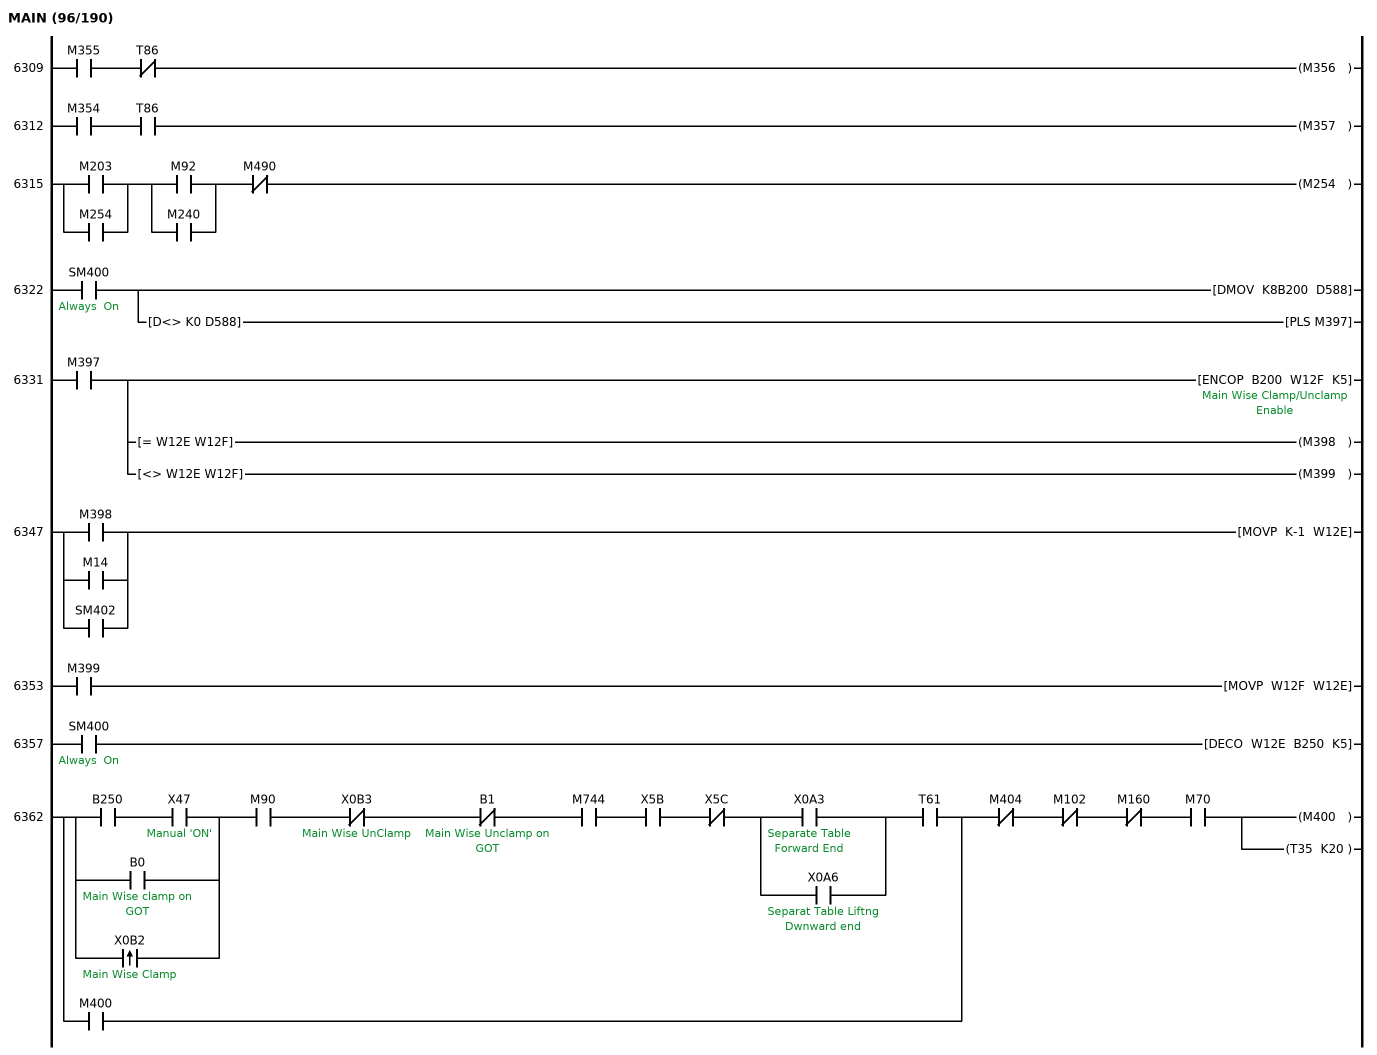
6309  LD      M355
      ANI     T86
      OUT     M356
6312  LD      M354
      AND     T86
      OUT     M357
6315  LD      M203
      OR      M254
      LD      M92
      OR      M240
      ANB
      ANI     M490
      OUT     M254
6322  LD      SM400  ; Always  On
      DMOV    K8B200 D588  ; Main Wise Clamp/Unclamp Enable
      ANDD<>  K0 D588
      PLS     M397
6331  LD      M397
      ENCOP   B200 W12F K5
      MPS
      AND=    W12E W12F
      OUT     M398
      MPP
      AND<>   W12E W12F
      OUT     M399
6347  LD      M398
      OR      M14
      OR      SM402
      MOVP    K-1 W12E
6353  LD      M399
      MOVP    W12F W12E
6357  LD      SM400  ; Always  On
      DECO    W12E B250 K5
6362  LD      B250
      AND     X47  ; Manual 'ON'
      OR      B0  ; Main Wise clamp on GOT
      ORP     X0B2  ; Main Wise Clamp
      AND     M90
      ANI     X0B3  ; Main Wise UnClamp
      ANI     B1  ; Main Wise Unclamp on GOT
      AND     M744
      AND     X5B
      ANI     X5C
      LD      X0A3  ; Separate Table Forward End
      OR      X0A6  ; Separat Table Liftng Dwnward end
      ANB
      AND     T61
      OR      M400
      ANI     M404
      ANI     M102
      ANI     M160
      AND     M70
      OUT     M400
      OUT     T35 K20
